FUNCTION_BLOCK FB_BHKW_Input
VAR_INPUT
	IN_Sammelstoerung		: BOOL;
END_VAR
VAR_OUTPUT
	Sammelstoerung			: BOOL;
END_VAR
VAR
END_VAR

Sammelstoerung := IN_Sammelstoerung;

END_FUNCTION_BLOCK

(* stored: Version 1.1.0.1, ProductVersion 3.1.4024.9
   POU FB_BHKW_Input: Id {e87c0bca-6793-4342-9c59-e14ffca6b131}, SpecialFunc None *)
